{attribute addProperty BoxType "EL3742-0000-0001"}
{attribute addProperty Id "Ch1_CycleCountAT %I*Ch1_CycleCount_2F207C3C1620Ch1_Sample_0AT %I*Ch1_Sample_37C07C831620Ch2_CycleCountAT %I*Ch2_CycleCount_7D759C541620Ch2_Sample_0AT %I*Ch2_Sample_29ECE4681620WcStateAT %I*WcState_C1B70B0F3240InfoDataAT %I*InfoData_7231B2DD80100"}
{attribute addProperty CRC "2345268208"}
{attribute addProperty SizeInBites "176"}
{attribute addProperty SizeInBytes "22"}
TYPE EL3742_FE433AD5 :
STRUCT
	{attribute addProperty Name "Ch1_CycleCount"}
	Ch1_CycleCount : Ch1_CycleCount_2F207C3C;
	{attribute addProperty Name "Ch1_Sample_0"}
	Ch1_Sample_0 : Ch1_Sample_37C07C83;
	{attribute addProperty Name "Ch2_CycleCount"}
	Ch2_CycleCount : Ch2_CycleCount_7D759C54;
	{attribute addProperty Name "Ch2_Sample_0"}
	Ch2_Sample_0 : Ch2_Sample_29ECE468;
	{attribute addProperty Name "WcState"}
	WcState : WcState_C1B70B0F;
	{attribute addProperty Name "InfoData"}
	InfoData : InfoData_7231B2DD;
END_STRUCT
END_TYPE

(* stored: Version 1.2.0.0, ProductVersion 3.1.4024.9
   DUT EL3742_FE433AD5: Id {fcbbe7da-748d-4fd9-b479-7582a38c40aa} *)
